// TIA Portal V16 export
// export: Created 2021-07-12T14:47:17.5325074Z, ExportSetting WithDefaults, DisplayName Totally Integrated Automation Portal, DisplayVersion V16, DisplayName TIA Portal Version Control Interface, DisplayVersion V16, DisplayName TIA Portal Openness, DisplayVersion V16, DisplayName STEP 7 Professional, DisplayVersion V16, DisplayName STEP 7 Safety, DisplayVersion V16, DisplayName WinCC Professional, DisplayVersion V16
VAR_GLOBAL   // PLC tag table "SimaHydTO_HydAxisAnalog_Interface"
   HydAxisAnalog_Sensor1_Interface_AddressIn AT %I1200.0 : "PD_TEL83_IN";   //    {ExternalWritable false}
   HydAxisAnalog_ForceSensor AT %IW1050 : Int;   //    {ExternalWritable false}
   HydAxisAnalog_Sensor1_Interface_AddressOut AT %Q1200.0 : "PD_TEL83_OUT";   //    {ExternalWritable false}
   HydAxisAnalog_OutputValue AT %QW0 : Int;   //    {ExternalWritable false}
END_VAR
